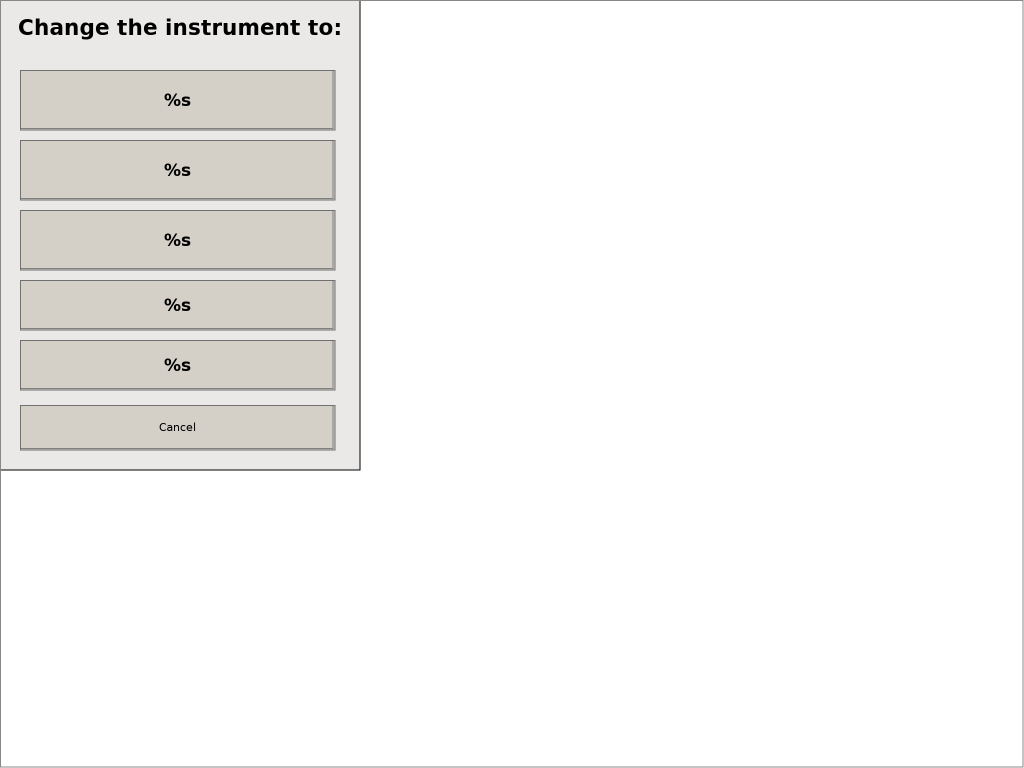
VISUALIZATION VISU_MTCSChangeInstrumentDialog  // 1024x768
    Rectangle (0,0 360x470)
    Button (20,70 315x60), "%s", text variable: GLOBAL.gui.changeInstrumentDialog.buttonsText[1], invisible if: GLOBAL.gui.changeInstrumentDialog.buttonsInvisible[1], input disabled if: GLOBAL.mtcs.processes.changeInstrument.statuses.enabledStatus.disabled
        OnMouseClick: execute { GLOBAL.gui.changeInstrumentDialog.buttonsDoRequest[1] := TRUE; }
        OnMouseClick: CloseDialog Dialog=VISU_MTCSChangeInstrumentDialog, Result=OK, NumpadKeypadSet=True
    Label (0,5 360x45), "Change the instrument to:"
    Button (20,405 315x45), "Cancel"
        OnMouseClick: CloseDialog Dialog=VISU_MTCSChangeInstrumentDialog, Result=OK, NumpadKeypadSet=True
    Button (20,140 315x60), "%s", text variable: GLOBAL.gui.changeInstrumentDialog.buttonsText[2], invisible if: GLOBAL.gui.changeInstrumentDialog.buttonsInvisible[2], input disabled if: GLOBAL.mtcs.processes.changeInstrument.statuses.enabledStatus.disabled
        OnMouseClick: execute { GLOBAL.gui.changeInstrumentDialog.buttonsDoRequest[2] := TRUE; }
        OnMouseClick: CloseDialog Dialog=VISU_MTCSChangeInstrumentDialog, Result=OK, NumpadKeypadSet=True
    Button (20,210 315x60), "%s", text variable: GLOBAL.gui.changeInstrumentDialog.buttonsText[3], invisible if: GLOBAL.gui.changeInstrumentDialog.buttonsInvisible[3], input disabled if: GLOBAL.mtcs.processes.changeInstrument.statuses.enabledStatus.disabled
        OnMouseClick: execute { GLOBAL.gui.changeInstrumentDialog.buttonsDoRequest[3] := TRUE; }
        OnMouseClick: CloseDialog Dialog=VISU_MTCSChangeInstrumentDialog, Result=OK, NumpadKeypadSet=True
    Button (20,280 315x50), "%s", text variable: GLOBAL.gui.changeInstrumentDialog.buttonsText[4], invisible if: GLOBAL.gui.changeInstrumentDialog.buttonsInvisible[4], input disabled if: GLOBAL.mtcs.processes.changeInstrument.statuses.enabledStatus.disabled
        OnMouseClick: execute { GLOBAL.gui.changeInstrumentDialog.buttonsDoRequest[4] := TRUE; }
        OnMouseClick: CloseDialog Dialog=VISU_MTCSChangeInstrumentDialog, Result=OK, NumpadKeypadSet=True
    Button (20,340 315x50), "%s", text variable: GLOBAL.gui.changeInstrumentDialog.buttonsText[5], invisible if: GLOBAL.gui.changeInstrumentDialog.buttonsInvisible[5], input disabled if: GLOBAL.mtcs.processes.changeInstrument.statuses.enabledStatus.disabled
        OnMouseClick: execute { GLOBAL.gui.changeInstrumentDialog.buttonsDoRequest[5] := TRUE; }
        OnMouseClick: CloseDialog Dialog=VISU_MTCSChangeInstrumentDialog, Result=OK, NumpadKeypadSet=True
END_VISUALIZATION

(* stored: Version 1.1.0.1, ProductVersion 3.1.4019.2
   Visu VISU_MTCSChangeInstrumentDialog: Id {4e53eae1-464b-4f39-8af5-2d4fb5bc2252} *)
